PROGRAM commandDecoder
VAR
	Command : STRING;
	Head_Loaded : STRING;
	Coordinate : WORD;
END_VAR

Command := F_ToLCase(GVL.stReceivedData);
GVL.stReceivedData := '';

//example
IF(Command = 'start') THEN
	Command := '';
	
ELSIF(Command = 'stop') THEN
	COM.doHome := FALSE;
	Command := '';
	
ELSIF(Command = 'home') THEN
	COM.doHome := TRUE;
	Command := '';
		
ELSE
	COM.doHome := FALSE; //temp
	Command := '';
	
END_IF;

END_PROGRAM

(* stored: Version 1.1.0.1, ProductVersion 3.1.4024.0
   POU commandDecoder: Id {7eba7217-46bb-46ef-8690-bb184ce360f6}, SpecialFunc None *)
